FUNCTION_BLOCK TemperatureInput EXTENDS AnalogInput
VAR_INPUT
END_VAR
VAR_OUTPUT
END_VAR
VAR
END_VAR
VAR PERSISTENT
END_VAR

SUPER^();
SignedWord := TRUE;

METHOD FB_init : BOOL
VAR_INPUT
	bInitRetains : BOOL; // if TRUE, the retain variables are initialized (warm start / cold start)
	bInCopyCode : BOOL;  // if TRUE, the instance afterwards gets moved into the copy code (online change)
END_VAR
IF bInitRetains THEN
	ProcessMin := -5000;
	ProcessMax := 15000;
	MinValue := -50;
	MaxValue := 150;
END_IF
END_METHOD

END_FUNCTION_BLOCK

(* stored: Version 1.1.0.1, ProductVersion 3.1.4024.6
   POU TemperatureInput: Id {24741fbc-de8f-4dad-9f51-c70e47fca627}, SpecialFunc None
   Method FB_init: Id {c18506e2-7257-4e6a-8e26-15b1532da28e} *)
